Yaskawa INFORM job: KRIS5NEW(-224_-90).JBI

/JOB
//NAME KRIS5NEW(-224_-90)
//POS
///NPOS 262,262,262,12,0,0
///TOOL 0
///POSTYPE PULSE
///PULSE
C00000=126,-73357,-105376,-18827,72039,-77556
C00001=32651,40852,-26417,-15259,84054,10521
C00002=30282,121459,21655,-7232,82256,-84550
C00003=119678,189491,121384,-6609,55844,-83781
C00004=119958,189291,121101,-6814,55937,-83682
C00005=119958,189291,121101,-6814,104918,-83682
C00006=69507,150313,105301,-6814,83622,-83682
C00007=102374,11647,-10601,-6208,113224,-88139
C00008=49110,-96581,-90191,-6208,113224,-88139
C00009=-73090,-118428,-105692,-6208,113224,-88139
C00010=-121621,-118428,-105692,-6208,113224,-88139
C00011=72199,118597,79738,-6814,89727,-83682
C00012=-14837,117754,79738,-6814,55937,-83682
C00013=-44504,100666,44561,-7265,69044,-83737
C00014=-106120,216,-72664,-1265,72875,-87293
C00015=-133015,-103640,-65816,3996,83698,-82063
C00016=-132086,-97485,-64003,4135,58701,-800
C00017=-87418,-103155,-50951,-24365,56592,18911
C00018=-91835,-92562,-47451,-18790,64201,15122
C00019=-91835,-90992,-44915,-18905,63486,15245
C00020=-91835,-91191,-45236,-18890,63577,15229
C00021=-92543,-89493,-44647,-18764,63906,14910
C00022=-91701,-93027,-47797,-18802,64208,15172
C00023=-103407,-97596,-50849,3072,56451,8420
C00024=-103441,-96475,-49251,3077,56046,8398
C00025=-103441,-95572,-47839,3092,55642,8386
C00026=-103441,-95784,-48170,3089,55737,8389
C00027=-103918,-93758,-47343,3170,56284,8224
C00028=-103441,-97091,-50215,3068,56323,8405
C00029=-109209,-114946,-61438,-11477,60008,8249
C00030=-109648,-104849,-49828,-11663,58030,8299
C00031=-106638,-101096,-45888,-12020,57948,9417
C00032=-106638,-99991,-44290,-12073,57541,9463
C00033=-106638,-100683,-45290,-12040,57795,9434
C00034=-107051,-98868,-44601,-11935,58240,9234
C00035=-106200,-104086,-48225,-12074,57912,9582
C00036=-152358,-99932,-47698,-5326,54954,-7442
C00037=-153713,-96711,-45144,-5074,54956,-7956
C00038=-153713,-95478,-43283,-5105,54446,-7931
C00039=-153713,-96622,-45010,-5076,54918,-7955
C00040=-152716,-94685,-44257,-5224,55508,-7607
C00041=-153713,-96622,-45010,-5076,54918,-7955
C00042=-147309,-120424,-63442,601,54974,-6742
C00043=-106734,-120076,-67764,3834,76101,81400
C00044=-118307,-107676,-53115,6964,73894,76814
C00045=-118315,-104761,-49202,6993,72991,76759
C00046=-118315,-103176,-46950,7014,72422,76727
C00047=-118315,-103373,-47231,7011,72492,76732
C00048=-118209,-105807,-47984,7053,71702,76722
C00049=-118315,-106666,-51906,6971,73669,76800
C00050=-152900,-100335,-49720,2405,77460,65790
C00051=-154432,-99514,-47530,2197,76577,65283
C00052=-154432,-98510,-46039,2200,76174,65277
C00053=-154432,-98792,-46458,2200,76287,65278
C00054=-155384,-100338,-46905,2069,75792,64965
C00055=-154432,-99810,-47974,2197,76697,65285
C00056=-139382,-109411,-63360,4215,80656,70261
C00057=-178843,-118258,-60230,-18880,61960,61638
C00058=-195730,-126290,-46968,-27647,52032,59296
C00059=-215647,-126319,-41034,-29483,43456,54148
C00060=-223903,-121672,-38076,-28785,41753,51233
C00061=-223903,-120259,-36425,-28941,41497,51327
C00062=-223903,-120713,-36957,-28890,41578,51297
C00063=-230177,-120958,-36962,-28394,39823,49171
C00064=-212196,-122715,-40198,-28895,45554,54842
C00065=-149200,-137053,-43419,-3768,60252,67444
C00066=-171288,-134336,-40679,-8987,58716,61402
C00067=-171288,-132312,-38502,-9016,58420,61427
C00068=-171288,-132787,-39014,-9009,58491,61421
C00069=-190720,-133903,-38866,-13381,55944,56165
C00070=-155339,-134276,-43064,-5179,61212,65702
C00071=-190109,-123977,-71374,-11222,85643,53403
C00072=-193209,-126845,-128640,-12422,104242,50582
C00073=-154889,-136514,-128640,-12422,104242,50582
C00074=49700,-188138,-128640,-12422,104242,50582
C00075=95044,-166675,-127403,-9604,101606,54242
C00076=100905,-121879,-41170,-2953,61354,-13811
C00077=76364,-126673,-37483,-7236,55371,-21106
C00078=76364,-125260,-35887,-7260,55120,-21085
C00079=76364,-125856,-36561,-7251,55227,-21092
C00080=80206,-125033,-36597,-6628,55913,-19986
C00081=76364,-128358,-39364,-7214,55663,-21122
C00082=106085,-127336,-41103,-2720,58495,-12699
C00083=106085,-125446,-38966,-2726,58152,-12693
C00084=106085,-125807,-39375,-2725,58219,-12694
C00085=107264,-124702,-39383,-2517,58821,-12358
C00086=106085,-127485,-41271,-2717,58524,-12702
C00087=100408,-120926,-37847,15529,71533,-19798
C00088=97019,-119074,-33059,14623,70083,-20929
C00089=97019,-117387,-31072,14654,69737,-20973
C00090=97019,-117741,-31491,14648,69810,-20964
C00091=98849,-116641,-31480,15187,70099,-20422
C00092=96336,-121085,-34976,14390,70314,-21090
C00093=117002,-126078,-36297,14353,59540,-14518
C00094=129547,-123648,-35340,18268,59922,-11292
C00095=117730,-128646,-41030,15406,62632,-14363
C00096=118409,-131302,-43968,5246,61629,-11067
C00097=120969,-131398,-38796,6988,54321,-10972
C00098=120206,-131306,-38746,6863,54384,-11194
C00099=120401,-140874,-53529,6577,58526,-10873
C00100=92949,-132183,-43651,2261,56631,-10244
C00101=85861,-128380,-38765,-239,57883,-11923
C00102=77238,-126478,-36922,-5379,55462,-19090
C00103=79359,-126575,-37043,-5049,55585,-18466
C00104=100444,-135554,-44697,-2672,56312,-10932
C00105=106086,-187684,-135216,-4534,68260,-4839
C00106=27739,-169745,-128413,-4049,68845,15832
C00107=-73947,-156826,-135344,-2505,79379,12508
C00108=-156474,-127565,-44757,-2910,70220,64434
C00109=-121984,-127790,-40571,3886,68541,67332
C00110=-112171,-127748,-37024,6888,65907,69854
C00111=-174367,-125221,-37157,-11588,65878,53298
C00112=-154263,-130476,-42112,2655,69883,62096
C00113=-147576,-136571,-44902,-18456,53984,64974
C00114=-183285,-124480,-40863,-3523,67329,53581
C00115=-173396,-130956,-37765,-24196,51014,58029
C00116=-177637,-130749,-37983,-24738,50343,56784
C00117=-142889,-132361,-46546,6897,66121,64856
C00118=-179390,-143866,-62624,-21295,53286,63054
C00119=-168678,-134236,-55921,-20538,56281,66231
C00120=-177027,-130604,-53028,-20333,54908,63602
C00121=-178065,-130378,-53013,-20352,54797,63256
C00122=-169128,-137015,-62017,-12044,61437,65819
C00123=-157938,-143674,-62364,-4171,59496,69325
C00124=-159280,-140899,-56089,-4426,57009,69004
C00125=-102188,-142365,-56060,2205,56882,86647
C00126=-106251,-146738,-64389,1676,59837,85440
C00127=-164064,-147455,-64185,5609,61717,65893
C00128=-130860,-150279,-64151,-6173,30547,-11978
C00129=-143649,-143019,-64547,-3233,38012,-18323
C00130=-155359,-132276,-57653,950,39168,-23559
C00131=-183290,-123860,-56538,17735,53089,-35896
C00132=-146679,-151365,-77655,-67,45404,-14364
C00133=-123624,-145278,-81119,-1216,58129,167
C00134=-124748,-141508,-71705,-1416,48370,-79
C00135=-109389,-139266,-70472,5539,48572,-999
C00136=-125400,-159913,-84219,1120,47581,-4556
C00137=-119711,-181360,-121572,-24950,66300,4723
C00138=-89347,-163256,-129350,-23289,87878,11502
C00139=-119711,-181360,-135603,-24950,39029,4723
C00140=-119711,-181360,-135603,-24950,39029,4723
C00141=-67118,-136665,-130676,-31892,63753,-5674
C00142=-40548,-161800,-132385,-30407,51173,2851
C00143=-38594,-160347,-135413,-37506,33521,-5777
C00144=-38158,-160025,-136084,-39080,61805,-7690
C00145=-9060,-155984,-136090,-36075,61852,-27249
C00146=-9060,-155984,-136090,-36075,61852,-27249
C00147=35778,-73357,-105376,-18827,72039,-77556
C00148=35778,-73357,-105376,-18827,72039,-77556
C00149=121972,-60692,-66036,-23906,48760,-72917
C00150=121972,-63565,-66036,-13351,77444,-72917
C00151=128597,-43861,-51514,-7611,79269,-70168
C00152=124571,-36839,-45278,-6435,81479,-71647
C00153=124571,-36774,-44033,-6444,80753,-71610
C00154=124571,-36787,-44229,-6442,80867,-71616
C00155=124620,-38693,-45447,-6456,80642,-71587
C00156=124571,-36854,-49289,-6406,83929,-71773
C00157=135784,-40512,-46259,8568,74966,-66573
C00158=131380,-30996,-39027,14250,80589,-67218
C00159=131380,-30921,-38010,14271,80021,-67284
C00160=131380,-30936,-38195,14267,80126,-67272
C00161=131516,-32861,-39482,14245,79911,-67249
C00162=128173,-31965,-42018,14869,82464,-68113
C00163=101589,-42073,-44271,32201,81327,-76893
C00164=104782,-94542,-85411,8339,74693,-77861
C00165=98731,-154827,-131308,9878,72678,-80158
C00166=98731,-154827,-131308,9878,72678,-80158
C00167=98731,-154827,-131308,9878,72678,-80158
C00168=141095,-137804,-121947,-4358,90462,-65341
C00169=171917,-153174,-112370,11397,78411,-54227
C00170=182434,-139119,-96629,10750,74982,-55468
C00171=188384,-139862,-92258,10800,71189,-53740
C00172=188384,-138592,-90710,10819,70894,-53767
C00173=188384,-138758,-90913,10816,70933,-53763
C00174=190704,-140607,-91317,10800,69944,-53044
C00175=183405,-135606,-91698,10796,73646,-55249
C00176=122437,-138897,-68678,7759,69704,-85075
C00177=122491,-138449,-67143,7802,68994,-85105
C00178=122491,-136911,-65445,7814,68742,-85121
C00179=122491,-137149,-65709,7813,68782,-85118
C00180=122596,-138957,-65891,7871,67964,-85140
C00181=122406,-137856,-68146,7745,69915,-85071
C00182=133908,-142665,-85466,-9447,80028,-78006
C00183=119924,-106608,-72308,-11523,88541,-83364
C00184=119912,-106121,-69782,-11526,87261,-83247
C00185=119912,-105140,-68125,-11527,86755,-83200
C00186=119912,-105255,-68320,-11527,86814,-83205
C00187=119890,-107421,-69006,-11532,86135,-83151
C00188=119921,-105912,-70668,-11522,87902,-83303
C00189=147950,-101609,-70952,8097,88078,-75282
C00190=148120,-101197,-69331,8117,87283,-75275
C00191=148120,-100369,-67808,8117,86776,-75308
C00192=148120,-100469,-67991,8117,86837,-75304
C00193=148835,-102702,-68752,8201,86094,-75111
C00194=147869,-101427,-71030,8086,88227,-75298
C00195=143601,-106428,-78314,14904,88558,-77172
C00196=127839,-150907,-89343,18520,59767,-2936
C00197=152748,-135569,-82180,5189,61325,8031
C00198=165584,-141067,-78434,-1748,48815,13484
C00199=165584,-139526,-76712,-1753,48546,13488
C00200=165584,-141067,-78434,-1748,48815,13484
C00201=163060,-138509,-78016,-1057,49832,12455
C00202=165969,-142680,-79869,-1849,48879,13638
C00203=102219,-150825,-81611,-4114,46497,-8124
C00204=103048,-146952,-79282,-4293,47091,-7814
C00205=103048,-145365,-77612,-4309,46878,-7806
C00206=103048,-146952,-79282,-4293,47091,-7814
C00207=104040,-144535,-78966,-4475,48184,-7463
C00208=103048,-146952,-79282,-4293,47091,-7814
C00209=130388,-156868,-90876,12327,55036,-1453
C00210=133185,-160601,-92679,12077,53862,-531
C00211=134262,-151926,-88228,13075,56181,-2073
C00212=134262,-150055,-86313,13106,55969,-2099
C00213=134262,-150290,-86556,13102,55997,-2095
C00214=133627,-147832,-86185,13029,57097,-2199
C00215=134630,-154151,-89309,13100,55659,-1999
C00216=134630,-154151,-89309,13100,55659,-1999
C00217=135665,-150111,-87290,12848,56320,-1524
C00218=135665,-148918,-86048,12870,56172,-1542
C00219=135665,-149404,-86555,12861,56233,-1535
C00220=135140,-147549,-86268,12816,57067,-1631
C00221=137258,-159588,-92377,12906,54393,-1161
C00222=125824,-157564,-85537,15505,47449,-6445
C00223=154464,-152435,-83956,11796,44323,4313
C00224=132203,-167713,-95137,7380,46601,51
C00225=129919,-160370,-92966,12704,53201,-3154
C00226=134642,-143084,-81504,11683,54346,-1201
C00227=125031,-149540,-76073,10907,40445,2143
C00228=120596,-149257,-75643,-12743,40882,6188
C00229=152241,-172921,-94343,-3507,40276,11220
C00230=158141,-110882,-79211,11782,79402,-69500
C00231=156021,-110302,-75029,11867,77473,-70419
C00232=159421,-110299,-72155,11937,75248,-69456
C00233=160676,-109631,-71837,11922,75213,-69024
C00234=131080,-121620,-80305,3109,79327,-78003
C00235=123808,-121005,-75422,2673,76894,-80480
C00236=107875,-120030,-75168,1641,77651,-85765
C00237=118816,-129868,-88464,-1274,80423,-81730
C00238=114341,-143568,-76470,-11022,70392,-81749
C00239=122142,-140123,-68459,-8102,68023,-79342
C00240=130964,-140542,-66172,-6885,67117,-76522
C00241=99704,-139575,-66025,-11086,64526,-86189
C00242=167439,-135845,-70174,10586,65898,-66819
C00243=173146,-130870,-67824,17958,62627,-66693
C00244=178018,-130516,-64419,18338,59826,-65420
C00245=178194,-130345,-64115,18355,59697,-65379
C00246=166403,-128472,-71093,17388,67046,-68381
C00247=164740,-137810,-91614,20635,72894,-68588
C00248=164740,-137810,-91614,20635,72894,-68588
C00249=149447,-191890,-120181,21381,67024,-75156
C00250=149584,-192173,-120256,21405,66899,-75131
C00251=149584,-192173,-120256,21405,66899,-75131
C00252=111536,-41528,-50064,5216,79386,-75344
C00253=113045,-31905,-41809,3207,85004,-74813
C00254=120280,-32752,-42293,1970,84637,-72395
C00255=120280,-32772,-45028,1968,86308,-72368
C00256=109334,-36848,-42541,23436,83058,-74194
C00257=110902,-28852,-35846,21774,87564,-72876
C00258=117885,-30007,-36632,20953,85658,-70699
C00259=109997,-31098,-41620,21879,90038,-72753
C00260=109380,-75662,-60137,33198,63885,-64520
C00261=9054,-143647,-113334,-5954,77551,-79151
BC00000=192636,515545,1075136
BC00001=106856,514699,1075147
BC00002=45026,513209,1075136
BC00003=297205,515545,1075136
BC00004=388258,132939,1075136
BC00005=388258,132939,1075136
BC00006=266781,91691,1075136
BC00007=338196,12076,1075135
BC00008=385019,2960,1075135
BC00009=385019,2960,1075135
BC00010=335835,2960,1075135
BC00011=245343,24956,1075136
BC00012=171885,-116810,981693
BC00013=145068,-168564,1075136
BC00014=282408,-168564,1075136
BC00015=324871,12764,1075136
BC00016=324871,12764,1033476
BC00017=324871,12764,1033476
BC00018=324871,12764,1033476
BC00019=324871,12764,1033476
BC00020=324871,12764,1033476
BC00021=324871,12764,1033476
BC00022=324871,12764,1033476
BC00023=342807,12764,1033476
BC00024=342807,12764,1033475
BC00025=342807,12764,1033475
BC00026=342807,12764,1033475
BC00027=342807,12764,1033475
BC00028=342807,12764,1033475
BC00029=324871,12764,1033476
BC00030=324871,12764,1033476
BC00031=324871,12764,1033476
BC00032=324871,12764,1033476
BC00033=324871,12764,1033476
BC00034=324871,12764,1033476
BC00035=324871,12764,1033476
BC00036=324871,12764,1033476
BC00037=324871,12764,1033476
BC00038=324871,12764,1033476
BC00039=324871,12764,1033476
BC00040=324871,12764,1033476
BC00041=324871,12764,1033476
BC00042=324871,12764,1033476
BC00043=324871,42664,1033476
BC00044=324871,42664,1033476
BC00045=324871,42664,1033476
BC00046=324871,42664,1033476
BC00047=324871,42664,1033476
BC00048=324871,42664,1033476
BC00049=324871,42664,1033476
BC00050=290678,42664,1033476
BC00051=290678,42664,1033476
BC00052=290678,42664,1033476
BC00053=290678,42664,1033476
BC00054=290678,42664,1033476
BC00055=290678,42664,1033476
BC00056=290678,42664,1033476
BC00057=324871,42664,1033476
BC00058=324871,70402,1033476
BC00059=324871,70402,1033476
BC00060=324871,70402,1033476
BC00061=324871,70402,1033476
BC00062=324871,70402,1033476
BC00063=324871,70402,1033476
BC00064=324871,70402,1033476
BC00065=339425,70402,1033476
BC00066=339425,70402,1033476
BC00067=339425,70402,1033476
BC00068=339425,70402,1033476
BC00069=339425,70402,1033476
BC00070=339425,70402,1033476
BC00071=338593,67759,1033476
BC00072=365604,66159,1034603
BC00073=365604,17709,1034603
BC00074=365604,1629,1034603
BC00075=299593,3037,1034603
BC00076=314294,3037,1034603
BC00077=328869,3461,1023592
BC00078=328869,3461,1023592
BC00079=328869,3461,1023592
BC00080=328869,3461,1023592
BC00081=328869,3461,1023592
BC00082=301345,10358,1012837
BC00083=301345,10358,1012837
BC00084=301345,10358,1012837
BC00085=301345,10358,1012837
BC00086=301345,10358,1012837
BC00087=302371,1302,1012837
BC00088=302371,1302,1012837
BC00089=302371,1302,1012837
BC00090=302371,1302,1012837
BC00091=302371,1302,1012837
BC00092=302371,1302,1012837
BC00093=302371,1302,1012837
BC00094=292881,1302,1012837
BC00095=310946,1302,1012837
BC00096=309160,1302,1012837
BC00097=309160,1302,1012837
BC00098=322422,1302,1012837
BC00099=322422,1302,1012837
BC00100=365717,2550,1012837
BC00101=365717,2550,1012837
BC00102=339278,3204,1020554
BC00103=325028,3204,1020554
BC00104=329399,3101,1025541
BC00105=344627,2742,1042919
BC00106=350887,22143,1073092
BC00107=276696,2854,1073092
BC00108=365604,67759,1033476
BC00109=338365,69290,1033476
BC00110=338365,69290,1033476
BC00111=338365,69290,1033476
BC00112=305385,71198,1033476
BC00113=309152,66398,1033476
BC00114=299083,59780,1033476
BC00115=307832,64230,1032960
BC00116=294760,64230,1032960
BC00117=299083,59780,1033476
BC00118=323021,86344,1018791
BC00119=323021,86344,1018791
BC00120=323021,86344,1018791
BC00121=309341,86344,1018791
BC00122=315244,86344,1018791
BC00123=339541,86344,1018791
BC00124=339541,86344,1018791
BC00125=339541,86344,1018791
BC00126=339541,86344,1018791
BC00127=320650,86344,1061699
BC00128=320650,38724,1061699
BC00129=296379,38724,988490
BC00130=296604,38724,988490
BC00131=348099,38724,988490
BC00132=348099,38724,988490
BC00133=331573,52292,963745
BC00134=331295,52292,963745
BC00135=358026,52292,963745
BC00136=350058,52292,963745
BC00137=317547,31600,963745
BC00138=278487,3584,1056780
BC00139=340345,-44387,1068891
BC00140=340345,-123490,1068891
BC00141=331767,-1766,1070081
BC00142=234698,5049,1063085
BC00143=254493,47555,1069374
BC00144=326806,106778,1070769
BC00145=344384,299723,1072198
BC00146=344384,446401,1072198
BC00147=295310,515545,1075136
BC00148=295310,513516,1075136
BC00149=295310,513263,813287
BC00150=335993,429318,731212
BC00151=335993,429318,731212
BC00152=335993,429318,731212
BC00153=335993,429318,731212
BC00154=335993,429318,731212
BC00155=335993,429318,731212
BC00156=335993,429318,731212
BC00157=327834,429318,731212
BC00158=327834,429318,731212
BC00159=327834,429318,731212
BC00160=327834,429318,731212
BC00161=327834,429318,731212
BC00162=327834,429318,731212
BC00163=292293,429318,731212
BC00164=292293,429318,731212
BC00165=292293,429318,979834
BC00166=314373,292172,979834
BC00167=314373,275872,695664
BC00168=349600,266255,695664
BC00169=349600,243768,695664
BC00170=339030,238977,762113
BC00171=339030,238977,762113
BC00172=339030,238977,762113
BC00173=339030,238977,762113
BC00174=339030,238977,762113
BC00175=339030,238977,762113
BC00176=351032,229664,891298
BC00177=351032,229664,891298
BC00178=351032,229664,891298
BC00179=351032,229664,891298
BC00180=351032,229664,891298
BC00181=351032,229664,891298
BC00182=326540,229664,891297
BC00183=314288,229664,891297
BC00184=314288,229664,891297
BC00185=314288,229664,891297
BC00186=314288,229664,891297
BC00187=314288,229664,891297
BC00188=314288,229664,891297
BC00189=310032,229664,891297
BC00190=310032,229664,891297
BC00191=310032,229664,891297
BC00192=310032,229664,891297
BC00193=310032,229664,891297
BC00194=310032,229664,891297
BC00195=317379,229664,891297
BC00196=317379,229664,891297
BC00197=343650,229664,891297
BC00198=343650,229664,891297
BC00199=343650,229664,891297
BC00200=343650,229664,891297
BC00201=343650,229664,891297
BC00202=343650,229664,891297
BC00203=343650,229664,891297
BC00204=343650,229664,891297
BC00205=343650,229664,891297
BC00206=343650,229664,891297
BC00207=343650,229664,891297
BC00208=343650,229664,891297
BC00209=323629,229664,891297
BC00210=263129,207424,891297
BC00211=263129,207424,891297
BC00212=263129,207424,891297
BC00213=263129,207424,891297
BC00214=263129,207424,891297
BC00215=263129,207424,891297
BC00216=327305,207424,891297
BC00217=327305,207424,891297
BC00218=327305,207424,891297
BC00219=327305,207424,891297
BC00220=327305,207424,891297
BC00221=327305,207424,891297
BC00222=327305,207424,891297
BC00223=267487,207457,891297
BC00224=287612,213644,891296
BC00225=310311,229663,891294
BC00226=310311,229663,891294
BC00227=310311,229663,891294
BC00228=360509,229663,891294
BC00229=334246,229663,891294
BC00230=310311,229663,891294
BC00231=337806,229663,891294
BC00232=336551,229663,891294
BC00233=323163,229663,891294
BC00234=337792,229663,891294
BC00235=337573,229663,891294
BC00236=337573,229663,891294
BC00237=310311,229663,891290
BC00238=308093,229663,891290
BC00239=320291,229663,891290
BC00240=320291,229663,891290
BC00241=320291,229663,891290
BC00242=335351,229663,891290
BC00243=335351,229663,891290
BC00244=335351,229663,891290
BC00245=320043,229663,891290
BC00246=320043,229663,891290
BC00247=335351,229663,891290
BC00248=352732,229663,1069777
BC00249=352732,229663,1069777
BC00250=352732,347909,1069777
BC00251=352732,347909,743295
BC00252=335993,429318,731212
BC00253=335993,429318,731212
BC00254=335993,429318,731212
BC00255=335993,429318,731212
BC00256=296648,426710,731211
BC00257=298029,426802,731211
BC00258=298029,426802,731211
BC00259=298029,426802,731211
BC00260=361465,487090,979283
BC00261=361465,516139,979283
EC00000=1986524,372644
EC00001=1986524,372644
EC00002=1986524,372644
EC00003=1986524,372644
EC00004=1986524,372644
EC00005=1986524,372644
EC00006=1986524,372644
EC00007=1986527,372644
EC00008=1986527,372644
EC00009=1986527,372644
EC00010=1986527,372644
EC00011=1986524,372644
EC00012=1986524,372644
EC00013=1986524,372644
EC00014=1986524,372644
EC00015=1986524,372644
EC00016=1986524,372644
EC00017=1986524,372644
EC00018=1986524,372644
EC00019=1986524,372644
EC00020=1986524,372644
EC00021=1986524,372644
EC00022=1986524,372644
EC00023=1986524,372644
EC00024=1986526,372644
EC00025=1986526,372644
EC00026=1986526,372644
EC00027=1986526,372644
EC00028=1986526,372644
EC00029=1986524,372644
EC00030=1986524,372644
EC00031=1986524,372644
EC00032=1986524,372644
EC00033=1986524,372644
EC00034=1986524,372644
EC00035=1986524,372644
EC00036=1986524,372644
EC00037=1986524,372644
EC00038=1986524,372644
EC00039=1986524,372644
EC00040=1986524,372644
EC00041=1986524,372644
EC00042=1986524,372644
EC00043=1986524,372644
EC00044=1986524,372644
EC00045=1986524,372644
EC00046=1986524,372644
EC00047=1986524,372644
EC00048=1986524,372644
EC00049=1986524,372644
EC00050=1986524,372644
EC00051=1986524,372644
EC00052=1986524,372644
EC00053=1986524,372644
EC00054=1986524,372644
EC00055=1986524,372644
EC00056=1986524,372644
EC00057=1986524,372644
EC00058=1986524,372644
EC00059=1986524,372644
EC00060=1986524,372644
EC00061=1986524,372644
EC00062=1986524,372644
EC00063=1986524,372644
EC00064=1986524,372644
EC00065=1986524,372644
EC00066=1986524,372644
EC00067=1986524,372644
EC00068=1986524,372644
EC00069=1986524,372644
EC00070=1986524,372644
EC00071=1986524,372644
EC00072=1986524,372644
EC00073=1986524,372644
EC00074=1986524,372644
EC00075=1986524,372644
EC00076=1986524,372644
EC00077=1986524,372644
EC00078=1986524,372644
EC00079=1986524,372644
EC00080=1986524,372644
EC00081=1986524,372644
EC00082=1986524,372644
EC00083=1986524,372644
EC00084=1986524,372644
EC00085=1986524,372644
EC00086=1986524,372644
EC00087=1986524,372644
EC00088=1986524,372644
EC00089=1986524,372644
EC00090=1986524,372644
EC00091=1986524,372644
EC00092=1986524,372644
EC00093=1986524,372644
EC00094=1986524,372644
EC00095=1986524,372644
EC00096=1986524,372644
EC00097=1986524,372644
EC00098=1986524,372644
EC00099=1986524,372644
EC00100=1986524,372644
EC00101=1986524,372644
EC00102=1986524,372644
EC00103=1986524,372644
EC00104=1986524,372644
EC00105=1986524,372644
EC00106=1986524,372644
EC00107=1986524,372644
EC00108=1986524,372644
EC00109=1986524,372644
EC00110=1986524,372644
EC00111=1986524,372644
EC00112=1986524,372644
EC00113=1986524,372644
EC00114=1986524,372644
EC00115=1986524,372644
EC00116=1986524,372644
EC00117=1986524,372644
EC00118=1986524,372644
EC00119=1986524,372644
EC00120=1986524,372644
EC00121=1986524,372644
EC00122=1986524,372644
EC00123=1986524,372644
EC00124=1986524,372644
EC00125=1986524,372644
EC00126=1986524,372644
EC00127=1986524,372644
EC00128=1986524,372644
EC00129=1986524,372644
EC00130=1986524,372644
EC00131=1986524,372644
EC00132=1986524,372644
EC00133=1986524,372644
EC00134=1986524,372644
EC00135=1986524,372644
EC00136=1986524,372644
EC00137=1986524,372644
EC00138=1986524,372644
EC00139=1986524,372644
EC00140=1986524,372644
EC00141=1924386,269829
EC00142=1942317,299498
EC00143=1898227,226544
EC00144=1888448,210364
EC00145=1813786,86826
EC00146=1813786,86826
EC00147=1660311,-167120
EC00148=1178646,-738387
EC00149=1144025,-740308
EC00150=1144025,-740308
EC00151=1144025,-740308
EC00152=1144025,-740308
EC00153=1144025,-740308
EC00154=1144025,-740308
EC00155=1144025,-740308
EC00156=1144025,-740308
EC00157=1144025,-740308
EC00158=1144025,-740308
EC00159=1144025,-740308
EC00160=1144025,-740308
EC00161=1144025,-740308
EC00162=1144025,-740308
EC00163=1144025,-740308
EC00164=1144025,-740308
EC00165=1144025,-740308
EC00166=1144025,-740308
EC00167=1144025,-740308
EC00168=1144025,-740308
EC00169=1144025,-740308
EC00170=1144025,-740308
EC00171=1144025,-740308
EC00172=1144025,-740308
EC00173=1144025,-740308
EC00174=1144025,-740308
EC00175=1144025,-740308
EC00176=1144025,-740308
EC00177=1144025,-740308
EC00178=1144025,-740308
EC00179=1144025,-740308
EC00180=1144025,-740308
EC00181=1144025,-740308
EC00182=1144023,-740308
EC00183=1144023,-740308
EC00184=1144023,-740308
EC00185=1144023,-740308
EC00186=1144023,-740308
EC00187=1144023,-740308
EC00188=1144023,-740308
EC00189=1144023,-740308
EC00190=1144023,-740308
EC00191=1144023,-740308
EC00192=1144023,-740308
EC00193=1144023,-740308
EC00194=1144023,-740308
EC00195=1144023,-740308
EC00196=1144023,-740308
EC00197=1144023,-740308
EC00198=1144023,-740308
EC00199=1144023,-740308
EC00200=1144023,-740308
EC00201=1144023,-740308
EC00202=1144023,-740308
EC00203=1144023,-740308
EC00204=1144023,-740308
EC00205=1144023,-740308
EC00206=1144023,-740308
EC00207=1144023,-740308
EC00208=1144023,-740308
EC00209=1144023,-740308
EC00210=1144023,-740308
EC00211=1144023,-740308
EC00212=1144023,-740308
EC00213=1144023,-740308
EC00214=1144023,-740308
EC00215=1144023,-740308
EC00216=1144023,-740308
EC00217=1144023,-740308
EC00218=1144023,-740308
EC00219=1144023,-740308
EC00220=1144023,-740308
EC00221=1144023,-740308
EC00222=1144023,-740308
EC00223=1144023,-740308
EC00224=1144022,-740308
EC00225=1144019,-740308
EC00226=1144019,-740308
EC00227=1144019,-740308
EC00228=1144019,-740308
EC00229=1144019,-740308
EC00230=1144019,-740308
EC00231=1144019,-740308
EC00232=1144019,-740308
EC00233=1144019,-740308
EC00234=1144019,-740308
EC00235=1144019,-740308
EC00236=1144019,-740308
EC00237=1144018,-740308
EC00238=1144018,-740308
EC00239=1144018,-740308
EC00240=1144018,-740308
EC00241=1144018,-740308
EC00242=1144018,-740308
EC00243=1144018,-740308
EC00244=1144018,-740308
EC00245=1144018,-740308
EC00246=1144018,-740308
EC00247=1144018,-740308
EC00248=1144018,-740308
EC00249=1144018,-740308
EC00250=1144018,-740308
EC00251=1144018,-740308
EC00252=1144025,-740308
EC00253=1144025,-740308
EC00254=1144025,-740308
EC00255=1144025,-740308
EC00256=1144023,-740309
EC00257=1144023,-740309
EC00258=1144023,-740309
EC00259=1144023,-740309
EC00260=1144023,-740309
EC00261=1207380,-740309
///POSTYPE BASE
///RECTAN
///RCONF 0,0,0,0,1,0,0,0,0,0,0,0,0,0,0,0,0,0,0,0,0,0,0,0
P00006=2.006,1.622,-0.565,0.0000,0.0000,0.0000
P00021=0.073,2.058,-0.109,0.0000,0.0000,0.0000
P00022=2.006,1.622,-0.565,0.0000,0.0000,0.0000
///RCONF 0,0,0,0,0,0,0,0,0,0,0,0,0,0,0,0,0,0,0,0,0,0,0,0
P00024=-1.466,-0.226,-0.419,0.0000,0.0000,0.0000
P00025=3.643,0.007,-2.585,0.0000,0.0000,0.0000
P00027=2.278,0.099,-4.210,0.0000,0.0000,0.0000
P00028=-1.778,-0.182,-2.050,0.0000,0.0000,0.0000
P00029=1.749,4.006,-0.261,0.0000,0.0000,0.0000
P00030=-0.014,-0.768,0.131,0.0000,0.0000,0.0000
P00031=-0.170,0.039,-0.647,0.0000,0.0000,0.0000
P00032=-0.423,0.157,3.222,0.0000,0.0000,0.0000
P00033=0.854,-1.099,3.047,0.0000,0.0000,0.0000
//INST
///DATE 2024/11/19 18:13
///ATTR SC,RW
///GROUP1 RB1,BS1
///GROUP2 ST1
NOP
'300124 MUZYLO
MOVJ C00000 BC00000 VJ=100.00  +MOVJ EC00000 VJ=100.00
CALL JOB:CLEAN-R1_KM_NEW
MOVJ C00001 BC00001 VJ=100.00  +MOVJ EC00001 VJ=100.00
MOVJ C00002 BC00002 VJ=100.00  +MOVJ EC00002 VJ=100.00
MOVJ C00003 BC00003 VJ=100.00  +MOVJ EC00003 VJ=100.00
MOVJ C00004 BC00004 VJ=100.00  +MOVJ EC00004 VJ=100.00
MOVJ C00005 BC00005 VJ=100.00  +MOVJ EC00005 VJ=0.78
MOVJ C00006 BC00006 VJ=100.00  +MOVJ EC00006 VJ=100.00
MOVJ C00007 BC00007 VJ=60.00  +MOVJ EC00007 VJ=60.00
MOVJ C00008 BC00008 VJ=60.00  +MOVJ EC00008 VJ=60.00
MOVJ C00009 BC00009 VJ=60.00  +MOVJ EC00009 VJ=60.00
MOVJ C00010 BC00010 VJ=60.00  +MOVJ EC00010 VJ=60.00
COMM MOVJ C00011 BC00011 VJ=100.00  +MOVJ EC00011 VJ=100.00
COMM MOVJ C00012 BC00012 VJ=100.00  +MOVJ EC00012 VJ=100.00
COMM MOVJ C00013 BC00013 VJ=100.00  +MOVJ EC00013 VJ=100.00
COMM MOVJ C00014 BC00014 VJ=100.00  +MOVJ EC00014 VJ=100.00
COMM MOVJ C00015 BC00015 VJ=100.00  +MOVJ EC00015 VJ=100.00
COMM MOVJ C00016 BC00016 VJ=100.00  +MOVJ EC00016 VJ=100.00
MOVJ C00017 BC00017 VJ=100.00  +MOVJ EC00017 VJ=100.00
SMOVL C00018 BC00018 V=100.0  +MOVJ EC00018
SREFP 3 C00019 BC00019  +REFP EC00019
CALL JOB:SEARCH-R1-S13D
SET P032 P006
SFTON3D P032
SMOVL C00020 BC00020 V=100.0  +MOVJ EC00020
SREFP 3 C00021 BC00021  +REFP EC00021
CALL JOB:SEARCH-R1-S13D
SET P032 P006
SFTON3D P032
SMOVL C00022 BC00022 V=100.0  +MOVJ EC00022
SFTOF3D
SMOVL C00023 BC00023 V=333.3  +MOVJ EC00023
SMOVL C00024 BC00024 V=100.0  +MOVJ EC00024
SREFP 3 C00025 BC00025  +REFP EC00025
CALL JOB:SEARCH-R1-S13D
SET P033 P006
SFTON3D P033
SMOVL C00026 BC00026 V=100.0  +MOVJ EC00026
SREFP 3 C00027 BC00027  +REFP EC00027
CALL JOB:SEARCH-R1-S13D
SET P033 P006
SFTON3D P033
SMOVL C00028 BC00028 V=100.0  +MOVJ EC00028
SFTOF3D
SMOVL C00029 BC00029 V=333.3  +MOVJ EC00029
SMOVL C00030 BC00030 V=1000.0  +MOVJ EC00030
SMOVL C00031 BC00031 V=100.0  +MOVJ EC00031
SREFP 3 C00032 BC00032  +REFP EC00032
CALL JOB:SEARCH-R1-S13D
SET P030 P006
SFTON3D P030
SMOVL C00033 BC00033 V=100.0  +MOVJ EC00033
SREFP 3 C00034 BC00034  +REFP EC00034
CALL JOB:SEARCH-R1-S13D
SET P030 P006
SFTON3D P030
SMOVL C00035 BC00035 V=100.0  +MOVJ EC00035
SFTOF3D
SMOVL C00036 BC00036 V=666.7  +MOVJ EC00036
SMOVL C00037 BC00037 V=100.0  +MOVJ EC00037
SREFP 3 C00038 BC00038  +REFP EC00038
CALL JOB:SEARCH-R1-S13D
SET P031 P006
SFTON3D P031
SMOVL C00039 BC00039 V=100.0  +MOVJ EC00039
SREFP 3 C00040 BC00040  +REFP EC00040
CALL JOB:SEARCH-R1-S13D
SET P031 P006
SFTON3D P031
SMOVL C00041 BC00041 V=100.0  +MOVJ EC00041
SFTOF3D
MOVJ C00042 BC00042 VJ=100.00  +MOVJ EC00042 VJ=100.00
MOVJ C00043 BC00043 VJ=100.00  +MOVJ EC00043 VJ=50.00
MOVJ C00044 BC00044 VJ=100.00  +MOVJ EC00044 VJ=50.00
SMOVL C00045 BC00045 V=100.0  +MOVJ EC00045
SREFP 3 C00046 BC00046  +REFP EC00046
CALL JOB:SEARCH-R1-S13D
SET P021 P006
SFTON3D P021
SMOVL C00047 BC00047 V=100.0  +MOVJ EC00047
SREFP 3 C00048 BC00048  +REFP EC00048
CALL JOB:SEARCH-R1-S13D
SET P021 P006
SFTON3D P021
SMOVL C00049 BC00049 V=100.0  +MOVJ EC00049
SFTOF3D
SMOVL C00050 BC00050 V=666.7  +MOVJ EC00050
SMOVL C00051 BC00051 V=100.0  +MOVJ EC00051
SREFP 3 C00052 BC00052  +REFP EC00052
CALL JOB:SEARCH-R1-S13D
SET P022 P006
SFTON3D P022
SMOVL C00053 BC00053 V=100.0  +MOVJ EC00053
SREFP 3 C00054 BC00054  +REFP EC00054
CALL JOB:SEARCH-R1-S13D
SET P022 P006
SFTON3D P022
SMOVL C00055 BC00055 V=100.0  +MOVJ EC00055
SFTOF3D
SMOVL C00056 BC00056 V=666.7  +MOVJ EC00056
SMOVL C00057 BC00057 V=333.3  +MOVJ EC00057
SMOVL C00058 BC00058 V=333.3  +MOVJ EC00058
SMOVL C00059 BC00059 V=333.3  +MOVJ EC00059
SMOVL C00060 BC00060 V=100.0  +MOVJ EC00060
SREFP 3 C00061 BC00061  +REFP EC00061
CALL JOB:SEARCH-R1-S13D
SET P024 P006
SFTON3D P024
SMOVL C00062 BC00062 V=100.0  +MOVJ EC00062
SREFP 3 C00063 BC00063  +REFP EC00063
CALL JOB:SEARCH-R1-S13D
SET P024 P006
SFTON3D P024
SMOVL C00064 BC00064 V=100.0  +MOVJ EC00064
SFTOF3D
SMOVL C00065 BC00065 V=666.7  +MOVJ EC00065
SMOVL C00066 BC00066 V=100.0  +MOVJ EC00066
SREFP 3 C00067 BC00067  +REFP EC00067
CALL JOB:SEARCH-R1-S13D
SET P025 P006
SFTON3D P025
SMOVL C00068 BC00068 V=100.0  +MOVJ EC00068
SREFP 3 C00069 BC00069  +REFP EC00069
CALL JOB:SEARCH-R1-S13D
SET P025 P006
SFTON3D P025
SMOVL C00070 BC00070 V=100.0  +MOVJ EC00070
SFTOF3D
MOVJ C00071 BC00071 VJ=100.00  +MOVJ EC00071 VJ=50.00
MOVJ C00072 BC00072 VJ=100.00  +MOVJ EC00072 VJ=50.00
MOVJ C00073 BC00073 VJ=60.00  +MOVJ EC00073 VJ=60.00
MOVJ C00074 BC00074 VJ=100.00  +MOVJ EC00074 VJ=50.00
MOVJ C00075 BC00075 VJ=60.00  +MOVJ EC00075 VJ=60.00
MOVJ C00076 BC00076 VJ=60.00  +MOVJ EC00076 VJ=60.00
SMOVL C00077 BC00077 V=166.7  +MOVJ EC00077
SREFP 3 C00078 BC00078  +REFP EC00078
CALL JOB:SEARCH-R1-S13D
SET P027 P006
SFTON3D P027
SMOVL C00079 BC00079 V=100.0  +MOVJ EC00079
SREFP 3 C00080 BC00080  +REFP EC00080
CALL JOB:SEARCH-R1-S13D
SET P027 P006
SFTON3D P027
SMOVL C00081 BC00081 V=166.7  +MOVJ EC00081
SFTOF3D
COMM SMOVL C00082 BC00082 V=100.0  +MOVJ EC00082
COMM SREFP 3 C00083 BC00083  +REFP EC00083
COMM CALL JOB:SEARCH-R1-S13D
COMM SET P028 P006
COMM SFTON3D P028
COMM SMOVL C00084 BC00084 V=100.0  +MOVJ EC00084
COMM SREFP 3 C00085 BC00085  +REFP EC00085
COMM CALL JOB:SEARCH-R1-S13D
COMM SET P028 P006
COMM SFTON3D P028
COMM SMOVL C00086 BC00086 V=100.0  +MOVJ EC00086
COMM SFTOF3D
COMM SMOVL C00087 BC00087 V=333.3  +MOVJ EC00087
COMM SMOVL C00088 BC00088 V=100.0  +MOVJ EC00088
COMM SREFP 3 C00089 BC00089  +REFP EC00089
COMM CALL JOB:SEARCH-R1-S13D
COMM SET P029 P006
COMM SFTON3D P029
COMM SMOVL C00090 BC00090 V=100.0  +MOVJ EC00090
COMM SREFP 3 C00091 BC00091  +REFP EC00091
COMM CALL JOB:SEARCH-R1-S13D
COMM SET P029 P006
COMM SFTON3D P029
COMM SMOVL C00092 BC00092 V=100.0  +MOVJ EC00092
COMM MACRO1 MJ#(0) ARGF14
COMM 'SPAWANIE 1CZ.
COMM SMOVL C00093 BC00093 V=133.3  +MOVJ EC00093
COMM ARCON
COMM SMOVL C00094 BC00094 V=10.0  +MOVJ EC00094
COMM ARCOF
COMM SFTOF3D
COMM SMOVL C00095 BC00095 V=250.0  +MOVJ EC00095
COMM SMOVL C00096 BC00096 V=500.0  +MOVJ EC00096
COMM SFTON3D P028
COMM SMOVL C00097 BC00097 V=166.7  +MOVJ EC00097
COMM ARCON
COMM SMOVL C00098 BC00098 V=10.0  +MOVJ EC00098
COMM ARCOF
COMM SFTOF3D
COMM SMOVL C00099 BC00099 V=166.7  +MOVJ EC00099
COMM SMOVL C00100 BC00100 V=666.7  +MOVJ EC00100
COMM SMOVL C00101 BC00101 V=83.3  +MOVJ EC00101
SFTON3D P027
SMOVL C00102 BC00102 V=83.3 PL=0  +MOVJ EC00102
ARCON
SMOVL C00103 BC00103 V=10.0  +MOVJ EC00103
ARCOF
SFTOF3D
SMOVL C00104 BC00104 V=166.7  +MOVJ EC00104
MOVJ C00105 BC00105 VJ=100.00  +MOVJ EC00105 VJ=50.00
MOVJ C00106 BC00106 VJ=100.00  +MOVJ EC00106 VJ=50.00
MOVJ C00107 BC00107 VJ=60.00  +MOVJ EC00107 VJ=60.00
MOVJ C00108 BC00108 VJ=50.00  +MOVJ EC00108 VJ=100.00
MOVL C00109 BC00109 V=250.0  +MOVJ EC00109 VJ=50.00
SFTON3D P025
SMOVL C00110 BC00110 V=133.3 PL=0  +MOVJ EC00110
ARCON
SMOVL C00111 BC00111 V=10.0  +MOVJ EC00111
ARCOF
SFTOF3D
SMOVL C00112 BC00112 V=166.7  +MOVJ EC00112
SMOVL C00113 BC00113 V=333.3  +MOVJ EC00113
SMOVL C00114 BC00114 V=166.7  +MOVJ EC00114
SFTON3D P024
SMOVL C00115 BC00115 V=166.7  +MOVJ EC00115
ARCON
SMOVL C00116 BC00116 V=10.0  +MOVJ EC00116
ARCOF
SFTOF3D
SMOVL C00117 BC00117 V=250.0  +MOVJ EC00117
SMOVL C00118 BC00118 V=250.0  +MOVJ EC00118
SMOVL C00119 BC00119 V=500.0  +MOVJ EC00119
SFTON3D P022
SMOVL C00120 BC00120 V=166.7  +MOVJ EC00120
ARCON
SMOVL C00121 BC00121 V=10.0  +MOVJ EC00121
ARCOF
SFTOF3D
SMOVL C00122 BC00122 V=500.0  +MOVJ EC00122
SMOVL C00123 BC00123 V=500.0  +MOVJ EC00123
SFTON3D P021
SMOVL C00124 BC00124 V=133.3 PL=0  +MOVJ EC00124
ARCON
SMOVL C00125 BC00125 V=10.0  +MOVJ EC00125
ARCOF
SFTOF3D
SMOVL C00126 BC00126 V=333.3  +MOVJ EC00126
MOVJ C00127 BC00127 VJ=100.00  +MOVJ EC00127 VJ=100.00
MOVJ C00128 BC00128 VJ=100.00  +MOVJ EC00128 VJ=100.00
MOVJ C00129 BC00129 VJ=100.00  +MOVJ EC00129 VJ=100.00
SFTON3D P031
SMOVL C00130 BC00130 V=166.7  +MOVJ EC00130
ARCON
SFTON3D P030
SMOVL C00131 BC00131 V=10.0  +MOVJ EC00131
ARCOF
SFTOF3D
SMOVL C00132 BC00132 V=250.0  +MOVJ EC00132
SMOVL C00133 BC00133 V=1000.0  +MOVJ EC00133
SFTON3D P032
SMOVL C00134 BC00134 V=166.7  +MOVJ EC00134
ARCON
SFTON3D P033
SMOVL C00135 BC00135 V=10.0  +MOVJ EC00135
ARCOF
SFTOF3D
SMOVL C00136 BC00136 V=500.0  +MOVJ EC00136
MOVJ C00137 BC00137 VJ=100.00  +MOVJ EC00137 VJ=30.00
MOVJ C00138 BC00138 VJ=100.00  +MOVJ EC00138 VJ=100.00
COMM MOVJ C00139 BC00139 VJ=100.00  +MOVJ EC00139 VJ=100.00
COMM MOVJ C00140 BC00140 VJ=100.00  +MOVJ EC00140 VJ=100.00
COMM MOVJ C00141 BC00141 VJ=100.00  +MOVJ EC00141 VJ=100.00
MOVJ C00142 BC00142 VJ=60.00  +MOVJ EC00142 VJ=60.00
MOVJ C00143 BC00143 VJ=60.00  +MOVJ EC00143 VJ=60.00
MOVJ C00144 BC00144 VJ=100.00  +MOVJ EC00144 VJ=100.00
MOVJ C00145 BC00145 VJ=20.00  +MOVJ EC00145 VJ=100.00
MOVJ C00146 BC00146 VJ=20.00  +MOVJ EC00146 VJ=20.00
'DRUGA POZYCJA
MOVJ C00147 BC00147 VJ=100.00  +MOVJ EC00147 VJ=100.00
MOVJ C00148 BC00148 VJ=100.00  +MOVJ EC00148 VJ=100.00
CALL JOB:CLEAN-R1_KM_NEW
MOVJ C00149 BC00149 VJ=100.00  +MOVJ EC00149 VJ=100.00
MOVJ C00150 BC00150 VJ=100.00  +MOVJ EC00150 VJ=100.00
MOVJ C00151 BC00151 VJ=100.00  +MOVJ EC00151 VJ=100.00
SMOVL C00152 BC00152 V=100.0  +MOVJ EC00152
SREFP 3 C00153 BC00153  +REFP EC00153
CALL JOB:SEARCH-R1-S13D
SET P021 P006
SFTON3D P021
SMOVL C00154 BC00154 V=100.0  +MOVJ EC00154
SREFP 3 C00155 BC00155  +REFP EC00155
CALL JOB:SEARCH-R1-S13D
SET P021 P006
SFTON3D P021
SMOVL C00156 BC00156 V=100.0  +MOVJ EC00156
SFTOF3D
SMOVL C00157 BC00157 V=333.3  +MOVJ EC00157
SMOVL C00158 BC00158 V=100.0  +MOVJ EC00158
SREFP 3 C00159 BC00159  +REFP EC00159
CALL JOB:SEARCH-R1-S13D
SET P022 P006
SFTON3D P022
SMOVL C00160 BC00160 V=100.0  +MOVJ EC00160
SREFP 3 C00161 BC00161  +REFP EC00161
CALL JOB:SEARCH-R1-S13D
SET P022 P006
SFTON3D P022
SMOVL C00162 BC00162 V=100.0  +MOVJ EC00162
SFTOF3D
SMOVL C00163 BC00163 V=333.3  +MOVJ EC00163
SMOVL C00164 BC00164 V=1000.0  +MOVJ EC00164
SMOVL C00165 BC00165 V=1000.0  +MOVJ EC00165
MOVJ C00166 BC00166 VJ=100.00  +MOVJ EC00166 VJ=100.00
MOVJ C00167 BC00167 VJ=100.00  +MOVJ EC00167 VJ=100.00
MOVJ C00168 BC00168 VJ=100.00  +MOVJ EC00168 VJ=100.00
MOVJ C00169 BC00169 VJ=100.00  +MOVJ EC00169 VJ=100.00
SMOVL C00170 BC00170 V=333.3  +MOVJ EC00170
SMOVL C00171 BC00171 V=100.0  +MOVJ EC00171
SREFP 3 C00172 BC00172  +REFP EC00172
CALL JOB:SEARCH-R1-S13D
SET P024 P006
SFTON3D P024
SMOVL C00173 BC00173 V=100.0  +MOVJ EC00173
SREFP 3 C00174 BC00174  +REFP EC00174
CALL JOB:SEARCH-R1-S13D
SET P024 P006
SFTON3D P024
SMOVL C00175 BC00175 V=100.0  +MOVJ EC00175
SFTOF3D
SMOVL C00176 BC00176 V=333.3  +MOVJ EC00176
SMOVL C00177 BC00177 V=100.0  +MOVJ EC00177
SREFP 3 C00178 BC00178  +REFP EC00178
CALL JOB:SEARCH-R1-S13D
SET P025 P006
SFTON3D P025
SMOVL C00179 BC00179 V=100.0  +MOVJ EC00179
SREFP 3 C00180 BC00180  +REFP EC00180
CALL JOB:SEARCH-R1-S13D
SET P025 P006
SFTON3D P025
SMOVL C00181 BC00181 V=100.0  +MOVJ EC00181
SFTOF3D
MOVJ C00182 BC00182 VJ=100.00  +MOVJ EC00182 VJ=50.00
MOVJ C00183 BC00183 VJ=100.00  +MOVJ EC00183 VJ=50.00
SMOVL C00184 BC00184 V=100.0  +MOVJ EC00184
SREFP 3 C00185 BC00185  +REFP EC00185
CALL JOB:SEARCH-R1-S13D
SET P027 P006
SFTON3D P027
SMOVL C00186 BC00186 V=100.0  +MOVJ EC00186
SREFP 3 C00187 BC00187  +REFP EC00187
CALL JOB:SEARCH-R1-S13D
SET P027 P006
SFTON3D P027
SMOVL C00188 BC00188 V=100.0  +MOVJ EC00188
SFTOF3D
SMOVL C00189 BC00189 V=250.0  +MOVJ EC00189
SMOVL C00190 BC00190 V=100.0  +MOVJ EC00190
SREFP 3 C00191 BC00191  +REFP EC00191
CALL JOB:SEARCH-R1-S13D
SET P028 P006
SFTON3D P028
SMOVL C00192 BC00192 V=100.0  +MOVJ EC00192
SREFP 3 C00193 BC00193  +REFP EC00193
CALL JOB:SEARCH-R1-S13D
SET P028 P006
SFTON3D P028
SMOVL C00194 BC00194 V=100.0  +MOVJ EC00194
SFTOF3D
MOVJ C00195 BC00195 VJ=100.00  +MOVJ EC00195 VJ=100.00
MOVJ C00196 BC00196 VJ=100.00  +MOVJ EC00196 VJ=100.00
MOVJ C00197 BC00197 VJ=100.00  +MOVJ EC00197 VJ=100.00
SMOVL C00198 BC00198 V=100.0  +MOVJ EC00198
SREFP 3 C00199 BC00199  +REFP EC00199
CALL JOB:SEARCH-R1-S13D
SET P030 P006
SFTON3D P030
SMOVL C00200 BC00200 V=100.0  +MOVJ EC00200
SREFP 3 C00201 BC00201  +REFP EC00201
CALL JOB:SEARCH-R1-S13D
SET P030 P006
SFTON3D P030
SMOVL C00202 BC00202 V=100.0  +MOVJ EC00202
SFTOF3D
SMOVL C00203 BC00203 V=416.7  +MOVJ EC00203
SMOVL C00204 BC00204 V=100.0  +MOVJ EC00204
SREFP 3 C00205 BC00205  +REFP EC00205
CALL JOB:SEARCH-R1-S13D
SET P031 P006
SFTON3D P031
SMOVL C00206 BC00206 V=100.0  +MOVJ EC00206
SREFP 3 C00207 BC00207  +REFP EC00207
CALL JOB:SEARCH-R1-S13D
SET P031 P006
SFTON3D P031
SMOVL C00208 BC00208 V=100.0  +MOVJ EC00208
SFTOF3D
SMOVL C00209 BC00209 V=500.0  +MOVJ EC00209
SMOVL C00210 BC00210 V=1000.0  +MOVJ EC00210
SMOVL C00211 BC00211 V=100.0  +MOVJ EC00211
SREFP 3 C00212 BC00212  +REFP EC00212
CALL JOB:SEARCH-R1-S13D
SET P033 P006
SFTON3D P033
SMOVL C00213 BC00213 V=100.0  +MOVJ EC00213
SREFP 3 C00214 BC00214  +REFP EC00214
CALL JOB:SEARCH-R1-S13D
SET P033 P006
SFTON3D P033
SMOVL C00215 BC00215 V=100.0  +MOVJ EC00215
SFTOF3D
SMOVL C00216 BC00216 V=416.7  +MOVJ EC00216
SMOVL C00217 BC00217 V=100.0  +MOVJ EC00217
SREFP 3 C00218 BC00218  +REFP EC00218
CALL JOB:SEARCH-R1-S13D
SET P032 P006
SFTON3D P032
SMOVL C00219 BC00219 V=100.0  +MOVJ EC00219
SREFP 3 C00220 BC00220  +REFP EC00220
CALL JOB:SEARCH-R1-S13D
SET P032 P006
SFTON3D P032
SMOVL C00221 BC00221 V=100.0  +MOVJ EC00221
MACRO1 MJ#(0) ARGF14
SMOVL C00222 BC00222 V=166.7  +MOVJ EC00222
ARCON
SFTON3D P033
SMOVL C00223 BC00223 V=9.2  +MOVJ EC00223
ARCOF
SFTOF3D
SMOVL C00224 BC00224 V=416.7  +MOVJ EC00224
SMOVL C00225 BC00225 V=1000.0  +MOVJ EC00225
SMOVL C00226 BC00226 V=416.7  +MOVJ EC00226
SFTON3D P030
SMOVL C00227 BC00227 V=133.3  +MOVJ EC00227
ARCON
SFTON3D P031
SMOVL C00228 BC00228 V=8.3  +MOVJ EC00228
ARCOF
SFTOF3D
SMOVL C00229 BC00229 V=416.7  +MOVJ EC00229
MOVJ C00230 BC00230 VJ=100.00  +MOVJ EC00230 VJ=100.00
MOVJ C00231 BC00231 VJ=100.00  +MOVJ EC00231 VJ=100.00
'BRAK POM SPR CZY OK
SFTON3D P028
SMOVL C00232 BC00232 V=133.3  +MOVJ EC00232
ARCON
MOVL C00233 BC00233 V=10.0  +MOVJ EC00233 VJ=15.00
ARCOF
SFTOF3D
MOVJ C00234 BC00234 VJ=100.00  +MOVJ EC00234 VJ=15.00
SFTON3D P027
SMOVL C00235 BC00235 V=133.3  +MOVJ EC00235
ARCON
SMOVL C00236 BC00236 V=10.0  +MOVJ EC00236
ARCOF
SFTOF3D
SMOVL C00237 BC00237 V=500.0  +MOVJ EC00237
SMOVL C00238 BC00238 V=250.0  +MOVJ EC00238
SFTON3D P025
SMOVL C00239 BC00239 V=250.0  +MOVJ EC00239
SMOVL C00240 BC00240 V=133.3  +MOVJ EC00240
ARCON
SMOVL C00241 BC00241 V=10.0  +MOVJ EC00241
ARCOF
SFTOF3D
SMOVL C00242 BC00242 V=250.0  +MOVJ EC00242
SMOVL C00243 BC00243 V=500.0  +MOVJ EC00243
SFTON3D P024
SMOVL C00244 BC00244 V=133.3  +MOVJ EC00244
ARCON
SMOVL C00245 BC00245 V=10.0  +MOVJ EC00245
ARCOF
SFTOF3D
SMOVL C00246 BC00246 V=666.7  +MOVJ EC00246
SMOVL C00247 BC00247 V=1000.0  +MOVJ EC00247
SMOVL C00248 BC00248 V=333.3  +MOVJ EC00248
SMOVL C00249 BC00249 V=1000.0  +MOVJ EC00249
SMOVL C00250 BC00250 V=1000.0  +MOVJ EC00250
SMOVL C00251 BC00251 V=1000.0  +MOVJ EC00251
SMOVL C00252 BC00252 V=666.7  +MOVJ EC00252
SFTON3D P021
SMOVL C00253 BC00253 V=133.3  +MOVJ EC00253
ARCON
SMOVL C00254 BC00254 V=10.0  +MOVJ EC00254
ARCOF
SFTOF3D
SMOVL C00255 BC00255 V=166.7  +MOVJ EC00255
SMOVL C00256 BC00256 V=666.7  +MOVJ EC00256
SFTON3D P022
SMOVL C00257 BC00257 V=133.3  +MOVJ EC00257
ARCON
SMOVL C00258 BC00258 V=10.0  +MOVJ EC00258
ARCOF
SFTOF3D
SMOVL C00259 BC00259 V=250.0  +MOVJ EC00259
MOVJ C00260 BC00260 VJ=100.00  +MOVJ EC00260 VJ=100.00
MOVJ C00261 BC00261 VJ=100.00  +MOVJ EC00261 VJ=100.00
END
